Fanuc KAREL source: kb00092.KL

-- PROVISIONAL review KL for V770-1; original PC SHA256 f4c9a9b461ff393492d0afc6024e70b5cc49eedc41a2eb3b10d62ed66c334334
-- Incomplete behavior may be omitted. Consult companion uncertainty JSON. Do not deploy.
PROGRAM KB00092
%NOLOCKGROUP
BEGIN
  -- UNRESOLVED_PC offsets 5-12; opcodes 9D,23
  -- UNRESOLVED_PC offsets 17-26; opcodes 3F,75
  -- UNRESOLVED_PC offsets 31-38; opcodes 9D,23
  -- UNRESOLVED_PC offsets 43-67; opcodes 27,22,22,2A,22,31
  -- UNRESOLVED_PC offsets 72-76; opcodes 7F
END KB00092
